// Mitsubishi GX Works2 project: HMI 연습 문제 코드 3   PLC: Q03UDV

PROGRAM MAIN
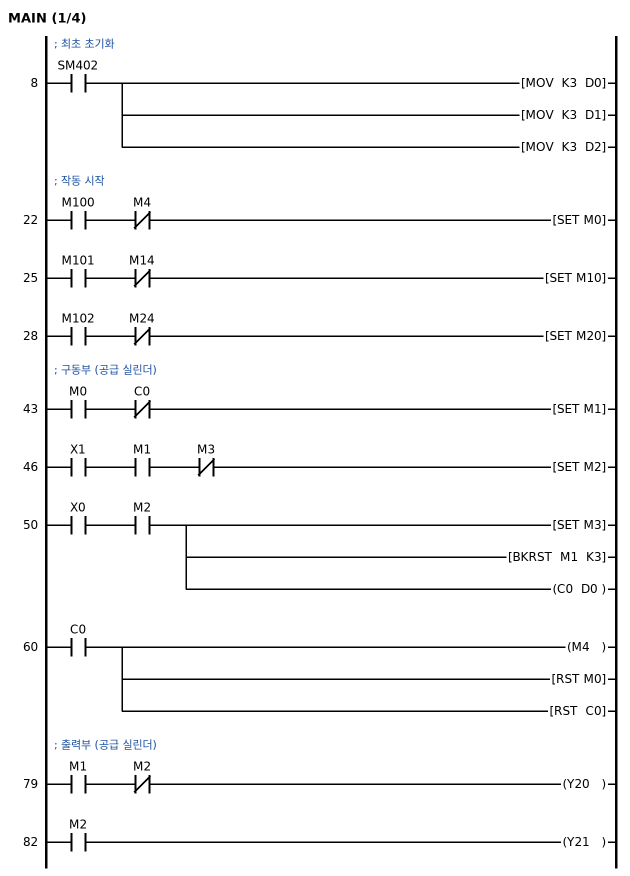
; 최초 초기화
8     LD      SM402
      MOV     K3 D0
      MOV     K3 D1
      MOV     K3 D2
; 작동 시작
22    LD      M100
      ANI     M4
      SET     M0
25    LD      M101
      ANI     M14
      SET     M10
28    LD      M102
      ANI     M24
      SET     M20
; 구동부 (공급 실린더)
43    LD      M0
      ANI     C0
      SET     M1
46    LD      X1
      AND     M1
      ANI     M3
      SET     M2
50    LD      X0
      AND     M2
      SET     M3
      BKRST   M1 K3
      OUT     C0 D0
60    LD      C0
      OUT     M4
      RST     M0
      RST     C0
; 출력부 (공급 실린더)
79    LD      M1
      ANI     M2
      OUT     Y20
82    LD      M2
      OUT     Y21
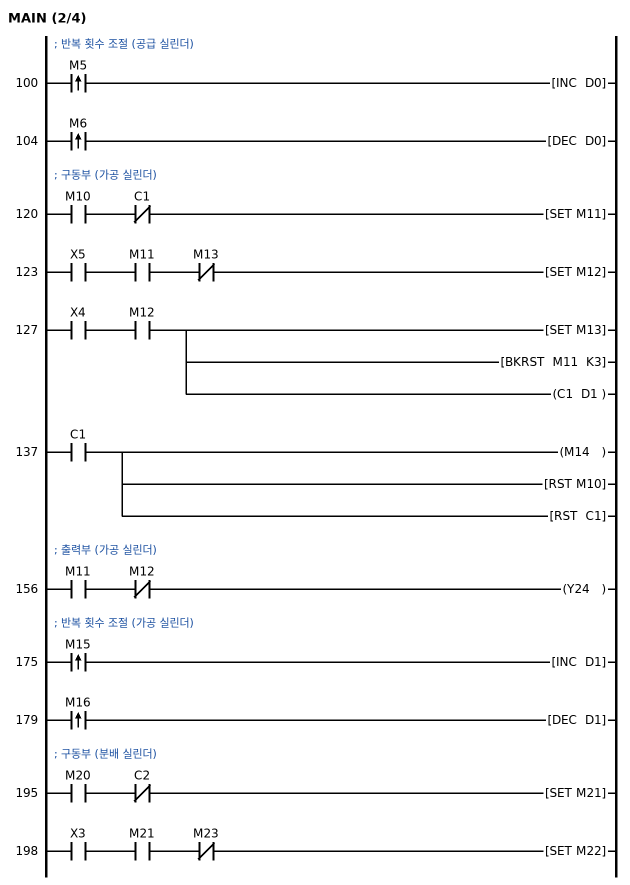
; 반복 횟수 조절 (공급 실린더)
100   LDP     M5
      INC     D0
104   LDP     M6
      DEC     D0
; 구동부 (가공 실린더)
120   LD      M10
      ANI     C1
      SET     M11
123   LD      X5
      AND     M11
      ANI     M13
      SET     M12
127   LD      X4
      AND     M12
      SET     M13
      BKRST   M11 K3
      OUT     C1 D1
137   LD      C1
      OUT     M14
      RST     M10
      RST     C1
; 출력부 (가공 실린더)
156   LD      M11
      ANI     M12
      OUT     Y24
; 반복 횟수 조절 (가공 실린더)
175   LDP     M15
      INC     D1
179   LDP     M16
      DEC     D1
; 구동부 (분배 실린더)
195   LD      M20
      ANI     C2
      SET     M21
198   LD      X3
      AND     M21
      ANI     M23
      SET     M22
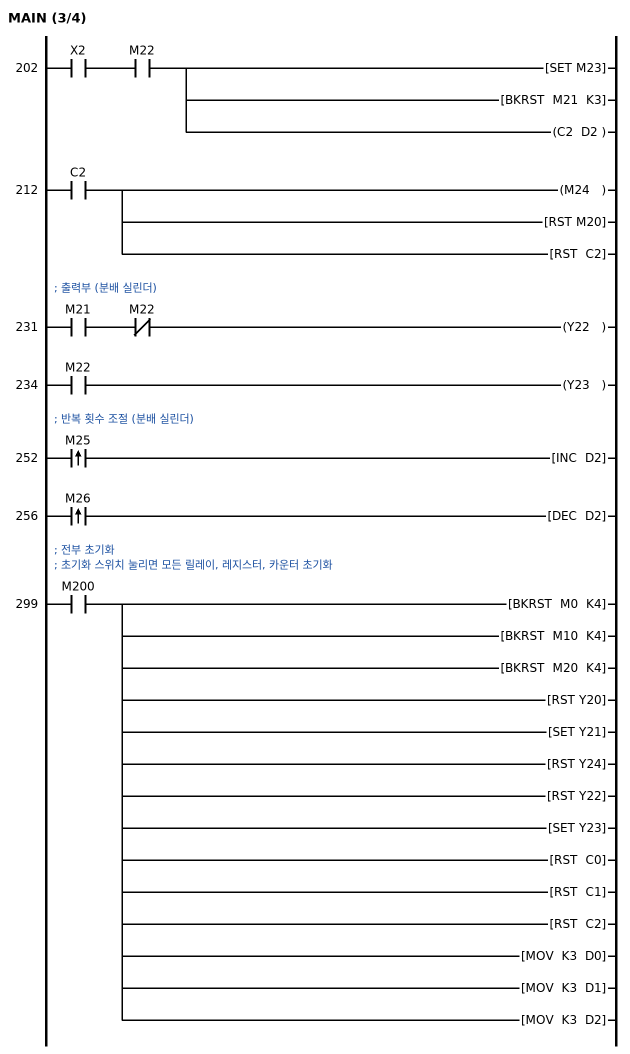
202   LD      X2
      AND     M22
      SET     M23
      BKRST   M21 K3
      OUT     C2 D2
212   LD      C2
      OUT     M24
      RST     M20
      RST     C2
; 출력부 (분배 실린더)
231   LD      M21
      ANI     M22
      OUT     Y22
234   LD      M22
      OUT     Y23
; 반복 횟수 조절 (분배 실린더)
252   LDP     M25
      INC     D2
256   LDP     M26
      DEC     D2
; 전부 초기화
; 초기화 스위치 눌리면 모든 릴레이, 레지스터, 카운터 초기화
299   LD      M200
      BKRST   M0 K4
      BKRST   M10 K4
      BKRST   M20 K4
      RST     Y20
      SET     Y21
      RST     Y24
      RST     Y22
      SET     Y23
      RST     C0
      RST     C1
      RST     C2
      MOV     K3 D0
      MOV     K3 D1
      MOV     K3 D2
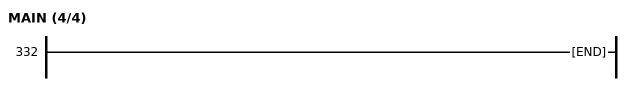
332   END
END_PROGRAM
